PROGRAM MAIN
VAR
  x : INT;
END_VAR

x := 1;

END_PROGRAM

(* stored: Version 1.0
   POU MAIN: Id {00000000-0000-0000-0000-000000000000} *)
